// TIA Portal V16 export
// export: Created 2023-01-04T15:44:09.0848348Z, ExportSetting WithDefaults, DisplayName Totally Integrated Automation Portal, DisplayVersion V16, DisplayName TIA Portal Version Control Interface, DisplayVersion V16, DisplayName TIA Portal Openness, DisplayVersion V16, DisplayName STEP 7 Professional, DisplayVersion V16, DisplayName STEP 7 Safety, DisplayVersion V16, DisplayName WinCC Advanced, DisplayVersion V16
DATA_BLOCK "Re-filling_Logic_DB"   // DB2
VERSION : 0.1
// stored: AutoNumber true, DBAccessibleFromOPCUA true, InstanceOfName Re-filling_Logic, InstanceOfType FB
"Re-filling_Logic"
BEGIN
END_DATA_BLOCK
